# EPICS substitutions: apps/mpodLvApp/Db/subs/fthodlv.substitutions
file "db/mpod8008l.db" {
    pattern {HOST,CH,SCAN,PORT,DETALIAS}
{"%(lvftag)","100","2 second","B_HW_LVFTAG_Sl1_Ch0","B_DET_FTH_LV_P"}
{"%(lvftag)","101","2 second","B_HW_LVFTAG_Sl1_Ch1","B_DET_FTH_LV_N"}
#{"%(lvftag)","102","2 second","B_HW_LVFTAG_Sl1_Ch2","B_DUMDUM_0"}
#{"%(lvftag)","103","2 second","B_HW_LVFTAG_Sl1_Ch3","B_DUMDUM_1"}
}
